KUKA KRL data list: HandEyeCalibrationExamp.dat

&ACCESS RVO
&REL 1
&PARAM DISKPATH = KRC:\R1\Program

DEFDAT HandEyeCalibrationExamp
   ;FOLD EXTERNAL DECLARATIONS;%{PE}%MKUKATPBASIS,%CEXT,%VCOMMON,%P
   ;FOLD BASISTECH EXT;%{PE}%MKUKATPBASIS,%CEXT,%VEXT,%P
   EXT  BAS (BAS_COMMAND  :IN,REAL  :IN )

   ;ENDFOLD (BASISTECH EXT)
   ;FOLD USER EXT;%{E}%MKUKATPUSER,%CEXT,%VEXT,%P
   ;Make your modifications here

   STRUC RETURNCODE_T INT VALUE,CHAR MSG[512]

   DECL INT RCEkiAliveFlagNo=997

   ;ENDFOLD (USER EXT)
   ;ENDFOLD (EXTERNAL DECLARATIONS)

   ; Teach following 8 hand eye calibration poses
   DECL E6POS XP1={X 0,Y 0,Z 0,A 0,B 0,C 0,S 0,T 0,E1 0.0,E2 0.0,E3 0.0,E4 0.0,E5 0.0,E6 0.0}
   DECL E6POS XP2={X 0,Y 0,Z 0,A 0,B 0,C 0,S 0,T 0,E1 0.0,E2 0.0,E3 0.0,E4 0.0,E5 0.0,E6 0.0}
   DECL E6POS XP3={X 0,Y 0,Z 0,A 0,B 0,C 0,S 0,T 0,E1 0.0,E2 0.0,E3 0.0,E4 0.0,E5 0.0,E6 0.0}
   DECL E6POS XP4={X 0,Y 0,Z 0,A 0,B 0,C 0,S 0,T 0,E1 0.0,E2 0.0,E3 0.0,E4 0.0,E5 0.0,E6 0.0}
   DECL E6POS XP5={X 0,Y 0,Z 0,A 0,B 0,C 0,S 0,T 0,E1 0.0,E2 0.0,E3 0.0,E4 0.0,E5 0.0,E6 0.0}
   DECL E6POS XP6={X 0,Y 0,Z 0,A 0,B 0,C 0,S 0,T 0,E1 0.0,E2 0.0,E3 0.0,E4 0.0,E5 0.0,E6 0.0}
   DECL E6POS XP7={X 0,Y 0,Z 0,A 0,B 0,C 0,S 0,T 0,E1 0.0,E2 0.0,E3 0.0,E4 0.0,E5 0.0,E6 0.0}
   DECL E6POS XP8={X 0,Y 0,Z 0,A 0,B 0,C 0,S 0,T 0,E1 0.0,E2 0.0,E3 0.0,E4 0.0,E5 0.0,E6 0.0}

   ; Declare the tool and base - Use a calibration grid tool for the HandEyeCalibration!
   DECL FDAT FP1={TOOL_NO 0,BASE_NO 0,IPO_FRAME #BASE,POINT2[] " "}

   DECL PDAT PPDAT1={VEL 20.0000,ACC 100.000,APO_DIST 500.000,APO_MODE #CDIS,GEAR_JERK 100.000,EXAX_IGN 0}

ENDDAT
